PROGRAM AppExample
VAR
	TcServer: TcTcpServer(BufferSize:= 1024);  // Receive buffer size per instance. Initialize the OTCID for the TcServer in the project instance
	Communication: CommunicationExample;
END_VAR

Communication(Server:= TcServer);  // Dependency inject the TcTcpServer implementation into the FB

END_PROGRAM

(* stored: Version 1.1.0.1
   POU AppExample: Id {03b40a06-ca0f-087c-3bcb-a70262e06c77}, SpecialFunc None *)
